Yaskawa INFORM job: K0.JBI

/JOB
//NAME K0
//POS
///NPOS 4,0,0,0
///TOOL 0
///PULSE
C000=-22857,32209,-30436,-145,-2762,-7062
C001=-21727,34313,-24907,2893,3896,-6692
C002=-19742,35411,-25844,-133,-3998,-7939
C003=-19492,35411,-26900,-133,-3998,-7939
//INST
///DATE 2014/09/30 23:39
///ATTR 0,0,0,0,0,0,0,0,0,0,0,0,0,1,0,0
///FRAME BASE
NOP
*1
MOVJ C000 VJ=25.00 PL=4
PAUSE
MOVJ C001 VJ=100.00 PL=4
MOVJ C002 VJ=100.00 PL=4
PAUSE
JUMP *1
MOVJ C003 VJ=100.00 CONT
END
